# EPICS autosave request: iocBoot/iocSimDetector/auto_settings.req
file "ADBase_settings.req", P=$(P), D=cam1:)
file "ADBase_settings.req", P=$(P), D=cam2:)
